// Mitsubishi GX Works2 project: 고속타이머   PLC: Q02/Q02H

PROGRAM MAIN
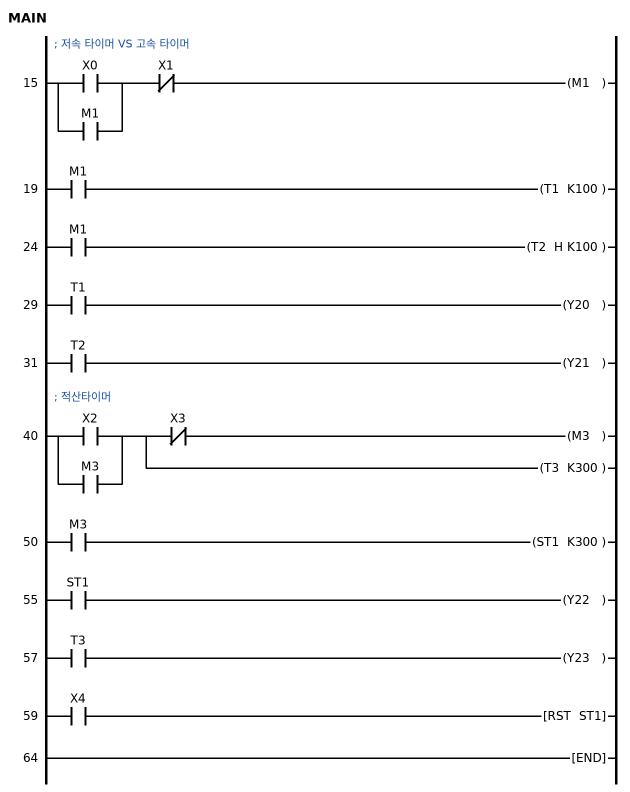
; 저속 타이머 VS 고속 타이머
15    LD      X0
      OR      M1
      ANI     X1
      OUT     M1
19    LD      M1
      OUT     T1 K100
24    LD      M1
      OUTH    T2 K100
29    LD      T1
      OUT     Y20
31    LD      T2
      OUT     Y21
; 적산타이머
40    LD      X2
      OR      M3
      MPS
      ANI     X3
      OUT     M3
      MPP
      OUT     T3 K300
50    LD      M3
      OUT     ST1 K300
55    LD      ST1
      OUT     Y22
57    LD      T3
      OUT     Y23
59    LD      X4
      RST     ST1
64    END
END_PROGRAM
